        rTestPosTop;
		TPWrite "Side 1 A";
		MoveJ pSafeS1, vmax, fine, tWeldGun\WObj:=wobjSide1A200;
		!Code Goes Here
		MoveJ pSafeS181, vmax, fine, tWeldGun\WObj:=wobjSide1A200;
		SingArea\Wrist;
		MoveJ [[1183.18,1457.45,363.98],[0.0635628,0.517234,-0.779105,0.348461],[0,1,-3,1],[9E+09,9E+09,9E+09,9E+09,9E+09,9E+09]], vmax, z10, tWeldGun\WObj:=wobjSide1A200;
		MoveL [[1181.95,1536.61,-4.61],[0.0635699,0.51724,-0.779104,0.348453],[0,1,-2,1],[9E+09,9E+09,9E+09,9E+09,9E+09,9E+09]], v1000, z10, tWeldGun\WObj:=wobjSide1A200;
		ArcLStart [[1183.34,1532.14,-10.38],[0.0432656,0.526366,-0.780926,0.333501],[0,1,-2,1],[9E+09,9E+09,9E+09,9E+09,9E+09,9E+09]], v10, seam13, weld13\Weave:=weave1, fine, tWeldGun\WObj:=wobjSide1A200;
		ArcLEnd [[1206.22,1532.24,-10.36],[0.0432175,0.526382,-0.780937,0.333453],[0,1,-2,1],[9E+09,9E+09,9E+09,9E+09,9E+09,9E+09]], v10, seam13, weld13\Weave:=weave1, fine, tWeldGun\WObj:=wobjSide1A200;
		MoveL [[1204.62,1537.22,-4.87],[0.0635798,0.517232,-0.779109,0.348451],[0,1,-2,1],[9E+09,9E+09,9E+09,9E+09,9E+09,9E+09]], vmax, z10, tWeldGun\WObj:=wobjSide1A200;
		MoveL [[863.66,1538.85,77.89],[0.0635666,0.517243,-0.779097,0.348464],[0,1,-2,1],[9E+09,9E+09,9E+09,9E+09,9E+09,9E+09]], vmax, z10, tWeldGun\WObj:=wobjSide1A200;
		MoveJ [[861.58,1461.21,260.09],[0.14949,-0.376148,-0.839997,-0.361347],[0,1,-1,1],[9E+09,9E+09,9E+09,9E+09,9E+09,9E+09]], vmax, z10, tWeldGun\WObj:=wobjSide1A200;
		MoveL [[863.22,1468.67,-10.11],[0.149522,-0.376221,-0.839963,-0.361336],[0,1,-1,1],[9E+09,9E+09,9E+09,9E+09,9E+09,9E+09]], v1000, z10, tWeldGun\WObj:=wobjSide1A200;
		ArcLStart [[866.37,1476.97,-12.05],[0.0874714,-0.401117,-0.850564,-0.328626],[0,1,-1,1],[9E+09,9E+09,9E+09,9E+09,9E+09,9E+09]], v10, seam13, weld13\Weave:=weave1, fine, tWeldGun\WObj:=wobjSide1A200;
		ArcLEnd [[894.17,1477.17,-12.05],[0.0874956,-0.401178,-0.850524,-0.328648],[0,1,-1,1],[9E+09,9E+09,9E+09,9E+09,9E+09,9E+09]], v10, seam13, weld13\Weave:=weave1, fine, tWeldGun\WObj:=wobjSide1A200;
		MoveL [[886.08,1463.03,-7.28],[0.149478,-0.376156,-0.840008,-0.361317],[0,1,-1,1],[9E+09,9E+09,9E+09,9E+09,9E+09,9E+09]], vmax, z10, tWeldGun\WObj:=wobjSide1A200;
		MoveJ [[863.35,1506.96,224.59],[0.0635605,0.517248,-0.779091,0.348471],[0,1,-2,1],[9E+09,9E+09,9E+09,9E+09,9E+09,9E+09]], vmax, z10, tWeldGun\WObj:=wobjSide1A200;
		MoveL [[863.49,1538.37,-7.85],[0.0635592,0.51724,-0.779122,0.348415],[0,1,-2,1],[9E+09,9E+09,9E+09,9E+09,9E+09,9E+09]], vmax, z10, tWeldGun\WObj:=wobjSide1A200;
		ArcLStart [[859.58,1532.06,-11.51],[0.0485275,0.53765,-0.768469,0.343561],[0,1,-2,1],[9E+09,9E+09,9E+09,9E+09,9E+09,9E+09]], v10, seam13, weld13\Weave:=weave1, fine, tWeldGun\WObj:=wobjSide1A200;
		ArcLEnd [[891.59,1532.36,-10.59],[0.0487409,0.513057,-0.792225,0.326766],[0,1,-2,1],[9E+09,9E+09,9E+09,9E+09,9E+09,9E+09]], v10, seam13, weld13\Weave:=weave1, fine, tWeldGun\WObj:=wobjSide1A200;
		MoveL [[887.77,1539.90,182.89],[0.0635615,0.517251,-0.779088,0.348474],[0,1,-2,1],[9E+09,9E+09,9E+09,9E+09,9E+09,9E+09]], vmax, z10, tWeldGun\WObj:=wobjSide1A200;
		MoveJ [[1182.52,1470.34,61.27],[0.149538,-0.376243,-0.839941,-0.361358],[0,1,-1,1],[9E+09,9E+09,9E+09,9E+09,9E+09,9E+09]], vmax, z10, tWeldGun\WObj:=wobjSide1A200;
		MoveL [[1181.55,1464.42,-9.30],[0.148332,-0.500326,-0.790399,-0.320847],[0,1,-1,1],[9E+09,9E+09,9E+09,9E+09,9E+09,9E+09]], v1000, z10, tWeldGun\WObj:=wobjSide1A200;
		ArcLStart [[1177.33,1473.60,-12.87],[0.148345,-0.500351,-0.790382,-0.320842],[0,1,-1,1],[9E+09,9E+09,9E+09,9E+09,9E+09,9E+09]], v10, seam13, weld13\Weave:=weave1, fine, tWeldGun\WObj:=wobjSide1A200;
		ArcLEnd [[1207.54,1473.57,-12.86],[0.148337,-0.500345,-0.790386,-0.320845],[0,1,-1,1],[9E+09,9E+09,9E+09,9E+09,9E+09,9E+09]], v10, seam13, weld13\Weave:=weave1, fine, tWeldGun\WObj:=wobjSide1A200;
		MoveL [[1206.87,1462.04,-3.48],[0.148351,-0.500349,-0.790363,-0.320889],[0,1,-1,1],[9E+09,9E+09,9E+09,9E+09,9E+09,9E+09]], vmax, z10, tWeldGun\WObj:=wobjSide1A200;
		MoveL [[1203.94,921.98,77.52],[0.149416,-0.376356,-0.839957,-0.361252],[0,1,-1,1],[9E+09,9E+09,9E+09,9E+09,9E+09,9E+09]], vmax, z10, tWeldGun\WObj:=wobjSide1A200;
		MoveL [[1209.28,920.32,-0.95],[0.0811338,-0.402507,-0.844244,-0.344469],[0,1,-1,1],[9E+09,9E+09,9E+09,9E+09,9E+09,9E+09]], v1000, z10, tWeldGun\WObj:=wobjSide1A200;
		ArcLStart [[1208.91,928.66,-10.99],[0.081096,-0.402552,-0.84423,-0.344458],[0,1,-1,1],[9E+09,9E+09,9E+09,9E+09,9E+09,9E+09]], v10, seam13, weld13\Weave:=weave1, fine, tWeldGun\WObj:=wobjSide1A200;
		ArcLEnd [[1180.12,929.43,-11.01],[0.0811029,-0.402583,-0.844212,-0.344465],[0,1,0,1],[9E+09,9E+09,9E+09,9E+09,9E+09,9E+09]], v10, seam13, weld13\Weave:=weave1, fine, tWeldGun\WObj:=wobjSide1A200;
		MoveL [[1182.60,918.33,-2.85],[0.0811745,-0.402551,-0.844212,-0.344485],[0,1,0,1],[9E+09,9E+09,9E+09,9E+09,9E+09,9E+09]], vmax, z10, tWeldGun\WObj:=wobjSide1A200;
		MoveL [[883.71,921.14,-1.64],[0.149424,-0.37639,-0.839933,-0.361269],[0,1,0,1],[9E+09,9E+09,9E+09,9E+09,9E+09,9E+09]], vmax, z10, tWeldGun\WObj:=wobjSide1A200;
		MoveL [[891.05,920.87,-4.97],[0.15161,-0.376469,-0.855824,-0.320705],[0,1,-1,1],[9E+09,9E+09,9E+09,9E+09,9E+09,9E+09]], v1000, z10, tWeldGun\WObj:=wobjSide1A200;
		ArcLStart [[890.95,930.44,-12.87],[0.151512,-0.376481,-0.855837,-0.320703],[0,1,-1,1],[9E+09,9E+09,9E+09,9E+09,9E+09,9E+09]], v10, seam13, weld13\Weave:=weave1, fine, tWeldGun\WObj:=wobjSide1A200;
		ArcLEnd [[864.65,932.03,-12.68],[0.151535,-0.376589,-0.85577,-0.320744],[0,1,-1,1],[9E+09,9E+09,9E+09,9E+09,9E+09,9E+09]], v10, seam13, weld13\Weave:=weave1, fine, tWeldGun\WObj:=wobjSide1A200;
		MoveL [[866.54,921.07,-4.87],[0.151523,-0.376433,-0.855874,-0.320656],[0,1,-1,1],[9E+09,9E+09,9E+09,9E+09,9E+09,9E+09]], v100, z10, tWeldGun\WObj:=wobjSide1A200;
		MoveL [[861.26,919.79,117.88],[0.149443,-0.376442,-0.8399,-0.361285],[0,1,-1,1],[9E+09,9E+09,9E+09,9E+09,9E+09,9E+09]], vmax, z0, tWeldGun\WObj:=wobjSide1A200;
		MoveJ [[868.17,991.07,127.71],[0.0426372,-0.330552,0.858067,-0.39069],[0,1,-2,1],[9E+09,9E+09,9E+09,9E+09,9E+09,9E+09]], vmax, z0, tWeldGun\WObj:=wobjSide1A200;
		MoveL [[863.71,988.79,-2.92],[0.042941,-0.330682,0.857982,-0.390734],[0,0,-2,1],[9E+09,9E+09,9E+09,9E+09,9E+09,9E+09]], v1000, z10, tWeldGun\WObj:=wobjSide1A200;
		ArcLStart [[861.89,984.77,-9.70],[0.0429638,-0.330722,0.857953,-0.39076],[0,0,-2,1],[9E+09,9E+09,9E+09,9E+09,9E+09,9E+09]], v10, seam13, weld13\Weave:=weave1, fine, tWeldGun\WObj:=wobjSide1A200;
		ArcLEnd [[898.10,985.21,-7.50],[0.0432219,-0.327548,0.859798,-0.389348],[0,0,-2,1],[9E+09,9E+09,9E+09,9E+09,9E+09,9E+09]], v10, seam13, weld13\Weave:=weave1, fine, tWeldGun\WObj:=wobjSide1A200;
		MoveL [[889.59,992.71,-6.61],[0.0430178,-0.330607,0.858002,-0.390745],[0,0,-2,1],[9E+09,9E+09,9E+09,9E+09,9E+09,9E+09]], vmax, z10, tWeldGun\WObj:=wobjSide1A200;
		MoveL [[889.59,992.73,75.52],[0.0430306,-0.330621,0.857997,-0.390743],[0,1,-2,1],[9E+09,9E+09,9E+09,9E+09,9E+09,9E+09]], vmax, z10, tWeldGun\WObj:=wobjSide1A200;
		MoveL [[1177.66,992.72,75.52],[0.0430182,-0.33062,0.857997,-0.390745],[0,0,-2,1],[9E+09,9E+09,9E+09,9E+09,9E+09,9E+09]], vmax, z10, tWeldGun\WObj:=wobjSide1A200;
		MoveL [[1185.35,990.20,-3.61],[0.0429073,-0.330578,0.858028,-0.390724],[0,0,-2,1],[9E+09,9E+09,9E+09,9E+09,9E+09,9E+09]], v1000, z10, tWeldGun\WObj:=wobjSide1A200;
		ArcLStart [[1176.08,984.61,-10.65],[0.0451953,-0.325527,0.859941,-0.390503],[0,0,-2,1],[9E+09,9E+09,9E+09,9E+09,9E+09,9E+09]], v10, seam13, weld13\Weave:=weave1, fine, tWeldGun\WObj:=wobjSide1A200;
		ArcLEnd [[1210.47,984.70,-10.67],[0.0451959,-0.325517,0.859949,-0.390493],[0,0,-2,1],[9E+09,9E+09,9E+09,9E+09,9E+09,9E+09]], v10, seam13, weld13\Weave:=weave1, fine, tWeldGun\WObj:=wobjSide1A200;
		MoveL [[1208.39,990.70,-6.82],[0.0442447,-0.330375,0.858404,-0.389919],[0,0,-2,1],[9E+09,9E+09,9E+09,9E+09,9E+09,9E+09]], v1000, z10, tWeldGun\WObj:=wobjSide1A200;
		MoveL [[1207.95,989.04,392.36],[0.0429563,-0.330627,0.857995,-0.39075],[0,1,-2,1],[9E+09,9E+09,9E+09,9E+09,9E+09,9E+09]], vmax, z10, tWeldGun\WObj:=wobjSide1A200;
		MoveJ [[194.09,1536.38,108.42],[0.0907205,-0.623393,0.712906,0.308084],[0,-1,0,1],[9E+09,9E+09,9E+09,9E+09,9E+09,9E+09]], vmax, z10, tWeldGun\WObj:=wobjSide1A200;
		MoveL [[194.09,1534.55,21.51],[0.0907097,-0.623392,0.712903,0.308096],[0,-1,0,1],[9E+09,9E+09,9E+09,9E+09,9E+09,9E+09]], vmax, z10, tWeldGun\WObj:=wobjSide1A200;
		ArcLStart [[190.35,1535.97,0.59],[0.0903662,-0.623335,0.713039,0.307999],[0,-1,0,1],[9E+09,9E+09,9E+09,9E+09,9E+09,9E+09]], v20, seam13, weld13\Weave:=weave1, fine, tWeldGun\WObj:=wobjSide1A200;
		ArcLEnd [[159.94,1535.93,0.55],[0.090343,-0.623341,0.713041,0.307988],[0,-1,0,1],[9E+09,9E+09,9E+09,9E+09,9E+09,9E+09]], v20, seam13, weld13\Weave:=weave1, fine, tWeldGun\WObj:=wobjSide1A200;
		MoveL [[158.09,1532.35,8.43],[0.0907075,-0.623402,0.712898,0.30809],[0,-1,0,1],[9E+09,9E+09,9E+09,9E+09,9E+09,9E+09]], vmax, z10, tWeldGun\WObj:=wobjSide1A200;
		MoveL [[-128.01,1535.58,7.69],[0.090663,-0.623378,0.712945,0.308043],[1,0,0,1],[9E+09,9E+09,9E+09,9E+09,9E+09,9E+09]], vmax, z10, tWeldGun\WObj:=wobjSide1A200;
		ArcLStart [[-127.83,1537.58,1.69],[0.0906477,-0.623383,0.712936,0.308058],[1,0,0,1],[9E+09,9E+09,9E+09,9E+09,9E+09,9E+09]], v20, seam13, weld13\Weave:=weave1, fine, tWeldGun\WObj:=wobjSide1A200;
		ArcLEnd [[-163.90,1538.90,1.91],[0.0906267,-0.6234,0.712927,0.308051],[1,0,0,1],[9E+09,9E+09,9E+09,9E+09,9E+09,9E+09]], v20, seam13, weld13\Weave:=weave1, fine, tWeldGun\WObj:=wobjSide1A200;
		SingArea\Wrist;
		MoveL [[-158.90,1535.32,931.69],[0.0906389,-0.623348,0.712932,0.308139],[1,-2,1,0],[9E+09,9E+09,9E+09,9E+09,9E+09,9E+09]], vmax, z0, tWeldGun\WObj:=wobjSide1A200;
		MoveJ [[-173.66,614.72,251.09],[0.128906,0.0495871,0.95885,-0.248055],[1,-1,1,0],[9E+09,9E+09,9E+09,9E+09,9E+09,9E+09]], vmax, z0, tWeldGun\WObj:=wobjSide1A200;
		MoveL [[-145.55,555.68,15.34],[0.152232,0.0392509,0.96562,-0.207034],[1,-1,1,0],[9E+09,9E+09,9E+09,9E+09,9E+09,9E+09]], vmax, z0, tWeldGun\WObj:=wobjSide1A200;
		ArcLStart [[-145.25,553.61,5.23],[0.150684,0.0446148,0.957996,-0.239891],[1,-1,1,0],[9E+09,9E+09,9E+09,9E+09,9E+09,9E+09]], v20, seam13, weld13\Weave:=weave1, fine, tWeldGun\WObj:=wobjSide1A200;
		ArcLEnd [[-113.04,553.61,5.21],[0.150682,0.0446047,0.957994,-0.239902],[1,-1,1,0],[9E+09,9E+09,9E+09,9E+09,9E+09,9E+09]], v20, seam13, weld13\Weave:=weave1, fine, tWeldGun\WObj:=wobjSide1A200;
		MoveL [[-113.65,555.41,12.33],[0.152159,0.0393397,0.96563,-0.207027],[1,-1,1,0],[9E+09,9E+09,9E+09,9E+09,9E+09,9E+09]], vmax, z0, tWeldGun\WObj:=wobjSide1A200;
		MoveL [[173.88,557.63,12.23],[0.150918,0.0436625,0.959445,-0.234057],[1,-1,1,0],[9E+09,9E+09,9E+09,9E+09,9E+09,9E+09]], vmax, z0, tWeldGun\WObj:=wobjSide1A200;
		ArcLStart [[173.75,552.63,2.66],[0.150938,0.0436659,0.959441,-0.234061],[1,-1,1,0],[9E+09,9E+09,9E+09,9E+09,9E+09,9E+09]], v20, seam13, weld13\Weave:=weave1, fine, tWeldGun\WObj:=wobjSide1A200;
		ArcLEnd [[207.36,552.81,2.26],[0.150944,0.0436531,0.959435,-0.234083],[1,-1,1,0],[9E+09,9E+09,9E+09,9E+09,9E+09,9E+09]], v20, seam13, weld13\Weave:=weave1, fine, tWeldGun\WObj:=wobjSide1A200;
		MoveL [[207.49,559.40,13.87],[0.152119,0.0394488,0.965633,-0.20702],[1,-1,1,0],[9E+09,9E+09,9E+09,9E+09,9E+09,9E+09]], vmax, z0, tWeldGun\WObj:=wobjSide1A200;
		MoveL [[862.60,554.49,14.86],[0.152154,0.0392658,0.965627,-0.207055],[0,-2,1,0],[9E+09,9E+09,9E+09,9E+09,9E+09,9E+09]], vmax, z0, tWeldGun\WObj:=wobjSide1A200;
		ArcLStart [[864.91,549.07,1.34],[0.133495,0.0503347,0.954435,-0.262108],[0,-1,1,0],[9E+09,9E+09,9E+09,9E+09,9E+09,9E+09]], v20, seam13, weld13\Weave:=weave1, fine, tWeldGun\WObj:=wobjSide1A200;
		ArcLEnd [[899.31,549.07,1.33],[0.133493,0.0503325,0.954436,-0.262103],[0,-2,1,0],[9E+09,9E+09,9E+09,9E+09,9E+09,9E+09]], v20, seam13, weld13\Weave:=weave1, fine, tWeldGun\WObj:=wobjSide1A200;
		MoveL [[899.33,555.62,9.82],[0.152106,0.0393027,0.965639,-0.207029],[0,-2,1,0],[9E+09,9E+09,9E+09,9E+09,9E+09,9E+09]], vmax, z0, tWeldGun\WObj:=wobjSide1A200;
		MoveL [[1178.47,554.50,11.88],[0.149638,0.047924,0.952344,-0.261443],[0,-2,1,0],[9E+09,9E+09,9E+09,9E+09,9E+09,9E+09]], vmax, z0, tWeldGun\WObj:=wobjSide1A200;
		ArcLStart [[1182.61,548.27,-0.41],[0.119114,0.0614783,0.947533,-0.290197],[0,-2,1,0],[9E+09,9E+09,9E+09,9E+09,9E+09,9E+09]], v20, seam13, weld13\Weave:=weave1, fine, tWeldGun\WObj:=wobjSide1A200;
		ArcLEnd [[1211.37,548.80,-1.22],[0.119109,0.0614608,0.947531,-0.290208],[0,-2,1,0],[9E+09,9E+09,9E+09,9E+09,9E+09,9E+09]], v20, seam13, weld13\Weave:=weave1, fine, tWeldGun\WObj:=wobjSide1A200;
		MoveL [[1185.29,583.76,320.77],[0.152081,0.0394165,0.965666,-0.206898],[0,-2,1,0],[9E+09,9E+09,9E+09,9E+09,9E+09,9E+09]], vmax, z0, tWeldGun\WObj:=wobjSide1A200;
		MoveJ [[759.22,820.77,477.02],[0.128857,0.0495447,0.958803,-0.24827],[0,-1,1,0],[9E+09,9E+09,9E+09,9E+09,9E+09,9E+09]], vmax, z0, tWeldGun\WObj:=wobjSide1A200;
		!legs start here
		MoveJ [[-401.88,982.38,420.80],[0.377905,-0.177501,-0.908663,-0.00353082],[1,0,1,0],[9E+09,9E+09,9E+09,9E+09,9E+09,9E+09]], vmax, z0, tWeldGun;
		MoveL [[-401.87,982.37,-5.96],[0.377901,-0.177501,-0.908665,-0.00352363],[1,0,1,0],[9E+09,9E+09,9E+09,9E+09,9E+09,9E+09]], v1000, z0, tWeldGun;
		ArcLStart [[-404.58,981.09,-7.78],[0.37795,-0.177396,-0.908665,-0.00362024],[1,0,1,0],[9E+09,9E+09,9E+09,9E+09,9E+09,9E+09]], v10, seam13, weld13\Weave:=weave1, fine, tWeldGun;
		ArcL [[-403.34,957.35,-6.28],[0.377997,-0.177583,-0.90861,-0.00339797],[1,0,1,0],[9E+09,9E+09,9E+09,9E+09,9E+09,9E+09]], v10, seam13, weld13\Weave:=weave1, z10, tWeldGun;
		ArcLEnd [[-425.46,950.14,-7.20],[0.197405,-0.679804,-0.668803,-0.227157],[1,0,2,0],[9E+09,9E+09,9E+09,9E+09,9E+09,9E+09]], v10, seam13, weld13\Weave:=weave1, fine, tWeldGun;
		MoveL [[-425.48,941.74,3.95],[0.197405,-0.679809,-0.668795,-0.227167],[1,0,2,0],[9E+09,9E+09,9E+09,9E+09,9E+09,9E+09]], vmax, z0, tWeldGun;
		MoveL [[-432.39,895.03,94.24],[0.274951,-0.581467,-0.743558,-0.182811],[1,0,2,0],[9E+09,9E+09,9E+09,9E+09,9E+09,9E+09]], vmax, z0, tWeldGun;
		MoveL [[-1101.20,895.02,94.24],[0.274939,-0.581469,-0.743563,-0.182805],[1,0,2,0],[9E+09,9E+09,9E+09,9E+09,9E+09,9E+09]], vmax, z0, tWeldGun;
		MoveL [[-1101.70,938.01,-1.40],[0.240452,-0.654006,-0.686015,-0.209388],[1,0,2,0],[9E+09,9E+09,9E+09,9E+09,9E+09,9E+09]], v1000, z0, tWeldGun;
		ArcLStart [[-1102.46,946.94,-5.88],[0.240345,-0.654194,-0.685887,-0.20934],[1,0,2,0],[9E+09,9E+09,9E+09,9E+09,9E+09,9E+09]], v10, seam13, weld13\Weave:=weave1, fine, tWeldGun;
		ArcL [[-1122.33,944.31,-5.63],[0.240415,-0.654059,-0.68597,-0.209414],[1,0,2,0],[9E+09,9E+09,9E+09,9E+09,9E+09,9E+09]], v10, seam13, weld13\Weave:=weave1, z10, tWeldGun;
		ArcLEnd [[-1131.87,975.46,-7.21],[0.0370294,0.922956,0.0834677,0.373919],[1,0,3,0],[9E+09,9E+09,9E+09,9E+09,9E+09,9E+09]], v10, seam13, weld13\Weave:=weave1, fine, tWeldGun;
		MoveL [[-1142.99,977.01,6.44],[0.0501214,0.923455,0.0523108,0.376805],[1,0,3,0],[9E+09,9E+09,9E+09,9E+09,9E+09,9E+09]], vmax, z0, tWeldGun;
		MoveJ [[-1224.84,979.29,303.50],[0.0444685,0.923113,0.0666376,0.376092],[1,0,-1,0],[9E+09,9E+09,9E+09,9E+09,9E+09,9E+09]], vmax, z20, tWeldGun;
		MoveL [[-1198.60,1154.71,4.46],[0.0444461,0.923123,0.0666424,0.37607],[1,0,-1,0],[9E+09,9E+09,9E+09,9E+09,9E+09,9E+09]], v1000, z0, tWeldGun;
		ArcLStart [[-1190.33,1151.56,-7.20],[0.0443887,0.92316,0.0665763,0.375997],[1,0,-1,0],[9E+09,9E+09,9E+09,9E+09,9E+09,9E+09]], v10, seam13, weld13\Weave:=weave1, fine, tWeldGun;
		ArcL [[-1193.47,1177.01,-8.64],[0.0444674,0.923156,0.0665468,0.376002],[1,0,-1,0],[9E+09,9E+09,9E+09,9E+09,9E+09,9E+09]], v10, seam13, weld13\Weave:=weave1, z10, tWeldGun;
		ArcLEnd [[-1167.22,1193.43,-4.61],[0.211529,0.696313,-0.654269,0.205758],[1,-1,0,0],[9E+09,9E+09,9E+09,9E+09,9E+09,9E+09]], v10, seam13, weld13\Weave:=weave1, fine, tWeldGun;
		MoveL [[-1165.81,1197.81,-4.44],[0.289046,0.665942,-0.622199,0.292988],[1,0,0,0],[9E+09,9E+09,9E+09,9E+09,9E+09,9E+09]], vmax, z0, tWeldGun;
		MoveL [[-1167.37,1197.80,267.48],[0.269054,0.631082,-0.684208,0.247398],[1,-1,0,0],[9E+09,9E+09,9E+09,9E+09,9E+09,9E+09]], vmax, z0, tWeldGun;
		MoveJ [[-491.85,1197.38,267.48],[0.269045,0.631086,-0.684208,0.247399],[1,-1,0,0],[9E+09,9E+09,9E+09,9E+09,9E+09,9E+09]], vmax, z0, tWeldGun;
		MoveL [[-493.75,1206.46,4.64],[0.230361,0.671978,-0.666396,0.226485],[1,-1,0,0],[9E+09,9E+09,9E+09,9E+09,9E+09,9E+09]], v1000, z0, tWeldGun;
		ArcLStart [[-496.53,1197.25,-8.21],[0.230282,0.672061,-0.666354,0.226445],[1,-1,0,0],[9E+09,9E+09,9E+09,9E+09,9E+09,9E+09]], v10, seam13, weld13\Weave:=weave1, fine, tWeldGun;
		ArcL [[-474.00,1197.10,-7.28],[0.230378,0.67197,-0.666403,0.226474],[1,-1,0,0],[9E+09,9E+09,9E+09,9E+09,9E+09,9E+09]], v10, seam13, weld13\Weave:=weave1, z10, tWeldGun;
		ArcLEnd [[-464.66,1164.90,-10.34],[0.384973,0.00807935,-0.922617,-0.0225858],[1,-1,1,0],[9E+09,9E+09,9E+09,9E+09,9E+09,9E+09]], v10, seam13, weld13\Weave:=weave1, fine, tWeldGun;
		MoveL [[-460.21,1166.10,-6.29],[0.384934,0.00803439,-0.922633,-0.0226006],[1,-1,1,0],[9E+09,9E+09,9E+09,9E+09,9E+09,9E+09]], vmax, z5, tWeldGun;
		MoveL [[-460.61,1166.13,158.38],[0.384913,0.00804793,-0.922641,-0.0226089],[1,-1,1,0],[9E+09,9E+09,9E+09,9E+09,9E+09,9E+09]], vmax, z5, tWeldGun;
		MoveJ [[-411.67,714.00,66.77],[0.262804,0.646065,-0.670013,0.254199],[1,-1,0,0],[9E+09,9E+09,9E+09,9E+09,9E+09,9E+09]], vmax, z5, tWeldGun;
		MoveL [[-412.17,719.36,-3.08],[0.242994,0.661127,-0.665052,0.248138],[1,-1,0,0],[9E+09,9E+09,9E+09,9E+09,9E+09,9E+09]], vmax, z5, tWeldGun;
		ArcLStart [[-411.16,714.15,-3.03],[0.22013,0.668771,-0.676855,0.214842],[1,-1,0,0],[9E+09,9E+09,9E+09,9E+09,9E+09,9E+09]], v5, seam13, weld13\Weave:=weave1, fine, tWeldGun;
		ArcLEnd [[-430.39,714.15,-6.45],[0.220118,0.668773,-0.67685,0.214862],[1,-1,0,0],[9E+09,9E+09,9E+09,9E+09,9E+09,9E+09]], v5, seam13, weld13\Weave:=weave1, fine, tWeldGun;
		MoveL [[-433.52,712.50,86.63],[0.256209,0.656106,-0.660016,0.261269],[1,-1,0,0],[9E+09,9E+09,9E+09,9E+09,9E+09,9E+09]], vmax, z5, tWeldGun;
		MoveL [[-1103.37,713.70,123.92],[0.256219,0.656103,-0.660014,0.261271],[1,-1,0,0],[9E+09,9E+09,9E+09,9E+09,9E+09,9E+09]], vmax, z5, tWeldGun;
		MoveL [[-1103.35,717.29,-4.25],[0.256222,0.656097,-0.66001,0.261295],[1,-1,0,0],[9E+09,9E+09,9E+09,9E+09,9E+09,9E+09]], vmax, z5, tWeldGun;
		ArcLStart [[-1103.12,713.69,-5.87],[0.256215,0.656125,-0.659976,0.261315],[1,-1,0,0],[9E+09,9E+09,9E+09,9E+09,9E+09,9E+09]], v5, seam13, weld13\Weave:=weave1, fine, tWeldGun;
		ArcLEnd [[-1131.44,712.83,-4.90],[0.256552,0.655237,-0.660527,0.261822],[1,-1,0,0],[9E+09,9E+09,9E+09,9E+09,9E+09,9E+09]], v5, seam13, weld13\Weave:=weave1, fine, tWeldGun;
		MoveL [[-1209.09,671.31,55.31],[0.0790996,-0.947264,0.00476783,-0.310504],[1,-1,-1,0],[9E+09,9E+09,9E+09,9E+09,9E+09,9E+09]], vmax, z5, tWeldGun;
		MoveJ [[-1174.22,1417.20,153.64],[0.288404,-0.63354,-0.657568,-0.288193],[1,-1,-2,0],[9E+09,9E+09,9E+09,9E+09,9E+09,9E+09]], vmax, z5, tWeldGun;
		MoveL [[-1161.88,1424.25,9.40],[0.288254,-0.633648,-0.657559,-0.288125],[1,-1,-2,0],[9E+09,9E+09,9E+09,9E+09,9E+09,9E+09]], vmax, z5, tWeldGun;
		ArcLStart [[-1160.66,1428.75,-9.26],[0.26399,-0.634491,-0.667287,-0.287158],[1,-1,-2,0],[9E+09,9E+09,9E+09,9E+09,9E+09,9E+09]], v5, seam13, weld13\Weave:=weave1, fine, tWeldGun;
		ArcLEnd [[-1185.26,1428.75,-8.26],[0.263991,-0.634496,-0.667282,-0.287157],[1,-1,-2,0],[9E+09,9E+09,9E+09,9E+09,9E+09,9E+09]], v5, seam13, weld13\Weave:=weave1, fine, tWeldGun;
		MoveL [[-1308.95,1421.25,86.72],[0.288384,-0.633585,-0.657536,-0.288188],[1,-1,-2,0],[9E+09,9E+09,9E+09,9E+09,9E+09,9E+09]], vmax, z5, tWeldGun;
		MoveL [[-494.06,1426.01,134.66],[0.280642,-0.634844,-0.656104,-0.296212],[1,-1,-2,0],[9E+09,9E+09,9E+09,9E+09,9E+09,9E+09]], vmax, z5, tWeldGun;
		MoveL [[-492.29,1429.04,-11.80],[0.251506,-0.647279,-0.667794,-0.268007],[1,-1,-2,0],[9E+09,9E+09,9E+09,9E+09,9E+09,9E+09]], vmax, z5, tWeldGun;
		ArcLStart [[-491.87,1429.46,-11.99],[0.251491,-0.647295,-0.667791,-0.267988],[1,-1,-2,0],[9E+09,9E+09,9E+09,9E+09,9E+09,9E+09]], v5, seam13, weld13\Weave:=weave1, fine, tWeldGun;
		ArcLEnd [[-476.29,1430.44,-11.13],[0.251464,-0.647334,-0.667765,-0.267984],[1,-1,-2,0],[9E+09,9E+09,9E+09,9E+09,9E+09,9E+09]], v5, seam13, weld13\Weave:=weave1, fine, tWeldGun;
		MoveL [[-335.43,1418.41,452.48],[0.280609,-0.634847,-0.656145,-0.296146],[1,-1,-2,0],[9E+09,9E+09,9E+09,9E+09,9E+09,9E+09]], vmax, z5, tWeldGun;
		MoveJ pSafeS1, vmax, fine, tWeldGun;

	ENDPROC

    PROC rRUNSide1A300()
        VAR num i;
            !300 Gallon Space Saver
           	rTestPosTop;
		TPWrite "Side 1 A";
        MoveJ pSafeS1, vmax, fine, tWeldGun;


            FOR i FROM 1 TO WeldiiiCount DO

                ! Optional safety check
                IF wp300{i}.start.trans.x <> 0 THEN
                    RunWeld(i);
                ENDIF

            ENDFOR
		MoveJ pSafeS1, vmax, fine, tWeldGun;
	ENDPROC

	PROC ss_200()
           	rTestPosTop;
		TPWrite "Side 1 A";
		MoveJ pSafeS1, vmax, fine, tWeldGun;
		!Code Goes Here
		MoveJ pSafeS181, vmax, fine, tWeldGun;
		SingArea\Wrist;
		MoveJ [[1181.97,1536.60,299.24],[0.0635588,0.517232,-0.779106,0.348462],[0,1,-3,1],[9E+09,9E+09,9E+09,9E+09,9E+09,9E+09]], vmax, z10, tWeldGun;
		MoveL [[1181.96,1536.60,-12.62],[0.0635661,0.517237,-0.779104,0.348458],[0,1,-2,1],[9E+09,9E+09,9E+09,9E+09,9E+09,9E+09]], v1000, z10, tWeldGun;
		ArcLStart [[1181.53,1529.02,-11.65],[0.0635714,0.517237,-0.779104,0.348457],[0,1,-2,1],[9E+09,9E+09,9E+09,9E+09,9E+09,9E+09]], v10, seam13, weld13\Weave:=weave1, fine, tWeldGun;
		ArcLEnd [[1204.96,1529.87,-10.62],[0.0635614,0.517237,-0.779103,0.348461],[0,1,-2,1],[9E+09,9E+09,9E+09,9E+09,9E+09,9E+09]], v10, seam13, weld13\Weave:=weave1, fine, tWeldGun;
		MoveL [[1204.64,1537.23,-12.62],[0.0635617,0.517239,-0.7791,0.348464],[0,1,-2,1],[9E+09,9E+09,9E+09,9E+09,9E+09,9E+09]], vmax, z10, tWeldGun;
		MoveL [[863.66,1538.85,77.89],[0.0635666,0.517243,-0.779097,0.348464],[0,1,-2,1],[9E+09,9E+09,9E+09,9E+09,9E+09,9E+09]], vmax, z10, tWeldGun;
		MoveJ [[861.58,1461.21,260.09],[0.14949,-0.376148,-0.839997,-0.361347],[0,1,-1,1],[9E+09,9E+09,9E+09,9E+09,9E+09,9E+09]], vmax, z10, tWeldGun;
		MoveL [[863.23,1471.68,-11.89],[0.149517,-0.37621,-0.839967,-0.361342],[0,1,-1,1],[9E+09,9E+09,9E+09,9E+09,9E+09,9E+09]], v1000, z10, tWeldGun;
		ArcLStart [[863.88,1474.96,-12.64],[0.149558,-0.376296,-0.839897,-0.361396],[0,1,-1,1],[9E+09,9E+09,9E+09,9E+09,9E+09,9E+09]], v10, seam13, weld13\Weave:=weave1, fine, tWeldGun;
		ArcLEnd [[887.67,1475.21,-13.25],[0.149548,-0.376266,-0.839942,-0.361327],[0,1,-1,1],[9E+09,9E+09,9E+09,9E+09,9E+09,9E+09]], v10, seam13, weld13\Weave:=weave1, fine, tWeldGun;
		MoveL [[886.08,1463.03,-7.28],[0.149478,-0.376156,-0.840008,-0.361317],[0,1,-1,1],[9E+09,9E+09,9E+09,9E+09,9E+09,9E+09]], vmax, z10, tWeldGun;
		MoveJ [[863.35,1506.96,224.59],[0.0635605,0.517248,-0.779091,0.348471],[0,1,-2,1],[9E+09,9E+09,9E+09,9E+09,9E+09,9E+09]], vmax, z10, tWeldGun;
		MoveL [[863.21,1535.55,-10.64],[0.0635626,0.51725,-0.779093,0.348463],[0,1,-2,1],[9E+09,9E+09,9E+09,9E+09,9E+09,9E+09]], vmax, z10, tWeldGun;
		ArcLStart [[862.98,1531.20,-11.14],[0.0635851,0.517245,-0.779094,0.348464],[0,1,-2,1],[9E+09,9E+09,9E+09,9E+09,9E+09,9E+09]], v10, seam13, weld13\Weave:=weave1, fine, tWeldGun;
		ArcLEnd [[887.38,1530.81,-10.94],[0.0635922,0.517251,-0.779089,0.348465],[0,1,-2,1],[9E+09,9E+09,9E+09,9E+09,9E+09,9E+09]], v10, seam13, weld13\Weave:=weave1, fine, tWeldGun;
		MoveL [[887.77,1539.90,182.89],[0.0635615,0.517251,-0.779088,0.348474],[0,1,-2,1],[9E+09,9E+09,9E+09,9E+09,9E+09,9E+09]], vmax, z10, tWeldGun;
		MoveJ [[1182.52,1470.34,61.27],[0.149538,-0.376243,-0.839941,-0.361358],[0,1,-1,1],[9E+09,9E+09,9E+09,9E+09,9E+09,9E+09]], vmax, z10, tWeldGun;
		MoveL [[1182.53,1470.34,-16.07],[0.149529,-0.376231,-0.83995,-0.361353],[0,1,-1,1],[9E+09,9E+09,9E+09,9E+09,9E+09,9E+09]], v1000, z10, tWeldGun;
		ArcLStart [[1181.99,1475.51,-15.52],[0.149552,-0.376279,-0.83992,-0.361363],[0,1,-1,1],[9E+09,9E+09,9E+09,9E+09,9E+09,9E+09]], v10, seam13, weld13\Weave:=weave1, fine, tWeldGun;
		ArcLEnd [[1204.38,1476.47,-15.60],[0.149569,-0.376356,-0.839878,-0.361375],[0,1,-1,1],[9E+09,9E+09,9E+09,9E+09,9E+09,9E+09]], v10, seam13, weld13\Weave:=weave1, fine, tWeldGun;
		MoveL [[1202.33,1469.98,-15.09],[0.149549,-0.376274,-0.839922,-0.361365],[0,1,-1,1],[9E+09,9E+09,9E+09,9E+09,9E+09,9E+09]], vmax, z10, tWeldGun;
		MoveL [[1203.94,921.98,77.52],[0.149416,-0.376356,-0.839957,-0.361252],[0,1,-1,1],[9E+09,9E+09,9E+09,9E+09,9E+09,9E+09]], vmax, z10, tWeldGun;
		MoveL [[1203.94,921.99,-12.97],[0.149422,-0.376348,-0.839957,-0.361259],[0,1,-1,1],[9E+09,9E+09,9E+09,9E+09,9E+09,9E+09]], v1000, z10, tWeldGun;
		ArcLStart [[1203.94,928.79,-14.21],[0.149423,-0.376362,-0.839952,-0.361256],[0,1,-1,1],[9E+09,9E+09,9E+09,9E+09,9E+09,9E+09]], v10, seam13, weld13\Weave:=weave1, fine, tWeldGun;
		ArcLEnd [[1178.19,928.79,-14.21],[0.149422,-0.376442,-0.839904,-0.361285],[0,1,-1,1],[9E+09,9E+09,9E+09,9E+09,9E+09,9E+09]], v10, seam13, weld13\Weave:=weave1, fine, tWeldGun;
		MoveL [[1177.78,921.50,-1.65],[0.149422,-0.376364,-0.839949,-0.36126],[0,1,-1,1],[9E+09,9E+09,9E+09,9E+09,9E+09,9E+09]], vmax, z10, tWeldGun;
		MoveL [[883.71,921.14,-1.64],[0.149424,-0.37639,-0.839933,-0.361269],[0,1,0,1],[9E+09,9E+09,9E+09,9E+09,9E+09,9E+09]], vmax, z10, tWeldGun;
		MoveL [[883.71,926.93,-12.24],[0.149423,-0.3764,-0.839927,-0.361273],[0,0,0,1],[9E+09,9E+09,9E+09,9E+09,9E+09,9E+09]], v1000, z10, tWeldGun;
		ArcLStart [[885.40,928.75,-13.38],[0.149454,-0.376503,-0.839867,-0.361295],[0,0,0,1],[9E+09,9E+09,9E+09,9E+09,9E+09,9E+09]], v10, seam13, weld13\Weave:=weave1, fine, tWeldGun;
		ArcLEnd [[866.41,928.73,-13.39],[0.149444,-0.376494,-0.839881,-0.361275],[0,0,0,1],[9E+09,9E+09,9E+09,9E+09,9E+09,9E+09]], v10, seam13, weld13\Weave:=weave1, fine, tWeldGun;
		MoveL [[863.70,926.54,-12.25],[0.149435,-0.37642,-0.839913,-0.361282],[0,0,0,1],[9E+09,9E+09,9E+09,9E+09,9E+09,9E+09]], v100, z10, tWeldGun;
		MoveL [[861.26,919.79,117.88],[0.149443,-0.376442,-0.8399,-0.361285],[0,1,-1,1],[9E+09,9E+09,9E+09,9E+09,9E+09,9E+09]], vmax, z0, tWeldGun;
		MoveJ [[868.17,991.07,127.71],[0.0426372,-0.330552,0.858067,-0.39069],[0,1,-2,1],[9E+09,9E+09,9E+09,9E+09,9E+09,9E+09]], vmax, z0, tWeldGun;
		MoveL [[868.52,991.54,-9.45],[0.0429862,-0.330642,0.857997,-0.390729],[0,0,-2,1],[9E+09,9E+09,9E+09,9E+09,9E+09,9E+09]], v1000, z10, tWeldGun;
		ArcLStart [[865.93,978.35,-10.52],[0.0429801,-0.330651,0.857991,-0.390736],[0,0,-2,1],[9E+09,9E+09,9E+09,9E+09,9E+09,9E+09]], v10, seam13, weld13\Weave:=weave1, fine, tWeldGun;
		ArcLEnd [[888.37,978.36,-11.00],[0.0429914,-0.330695,0.857973,-0.390738],[0,0,-2,1],[9E+09,9E+09,9E+09,9E+09,9E+09,9E+09]], v10, seam13, weld13\Weave:=weave1, fine, tWeldGun;
		MoveL [[889.59,992.71,-9.41],[0.0430222,-0.330607,0.858002,-0.390746],[0,0,-2,1],[9E+09,9E+09,9E+09,9E+09,9E+09,9E+09]], vmax, z10, tWeldGun;
		MoveL [[889.59,992.73,75.52],[0.0430306,-0.330621,0.857997,-0.390743],[0,1,-2,1],[9E+09,9E+09,9E+09,9E+09,9E+09,9E+09]], vmax, z10, tWeldGun;
		MoveL [[1177.66,992.72,75.52],[0.0430182,-0.33062,0.857997,-0.390745],[0,0,-2,1],[9E+09,9E+09,9E+09,9E+09,9E+09,9E+09]], vmax, z10, tWeldGun;
		MoveL [[1185.41,992.70,-11.53],[0.0429716,-0.330606,0.858007,-0.390739],[0,0,-2,1],[9E+09,9E+09,9E+09,9E+09,9E+09,9E+09]], v1000, z10, tWeldGun;
		ArcLStart [[1180.66,978.10,-13.63],[0.0429557,-0.330625,0.857997,-0.390747],[0,0,-2,1],[9E+09,9E+09,9E+09,9E+09,9E+09,9E+09]], v10, seam13, weld13\Weave:=weave1, fine, tWeldGun;
		ArcLEnd [[1207.05,977.71,-13.62],[0.0429527,-0.330628,0.857994,-0.390751],[0,0,-2,1],[9E+09,9E+09,9E+09,9E+09,9E+09,9E+09]], v10, seam13, weld13\Weave:=weave1, fine, tWeldGun;
		MoveL [[1207.94,989.04,-11.16],[0.0429397,-0.330625,0.858002,-0.39074],[0,0,-2,1],[9E+09,9E+09,9E+09,9E+09,9E+09,9E+09]], v1000, z10, tWeldGun;
		MoveL [[1207.95,989.04,392.36],[0.0429563,-0.330627,0.857995,-0.39075],[0,1,-2,1],[9E+09,9E+09,9E+09,9E+09,9E+09,9E+09]], vmax, z10, tWeldGun;
		MoveJ [[194.09,1536.38,108.42],[0.0907205,-0.623393,0.712906,0.308084],[0,-1,0,1],[9E+09,9E+09,9E+09,9E+09,9E+09,9E+09]], vmax, z10, tWeldGun;
		MoveL [[194.09,1534.55,44.51],[0.0907126,-0.623398,0.712901,0.308089],[0,-1,0,1],[9E+09,9E+09,9E+09,9E+09,9E+09,9E+09]], vmax, z10, tWeldGun;
		ArcLStart [[191.25,1532.54,0.05],[0.0904838,-0.623408,0.712969,0.30798],[0,-1,0,1],[9E+09,9E+09,9E+09,9E+09,9E+09,9E+09]], v20, seam13, weld13\Weave:=weave1, fine, tWeldGun;
		ArcLEnd [[157.22,1532.54,0.51],[0.090482,-0.623409,0.712967,0.307981],[0,-1,0,1],[9E+09,9E+09,9E+09,9E+09,9E+09,9E+09]], v20, seam13, weld13\Weave:=weave1, fine, tWeldGun;
		MoveL [[158.09,1532.35,8.43],[0.0907075,-0.623402,0.712898,0.30809],[0,-1,0,1],[9E+09,9E+09,9E+09,9E+09,9E+09,9E+09]], vmax, z10, tWeldGun;
		MoveL [[-123.91,1535.35,12.43],[0.0907124,-0.623396,0.712903,0.308089],[1,0,0,1],[9E+09,9E+09,9E+09,9E+09,9E+09,9E+09]], vmax, z10, tWeldGun;
		ArcLStart [[-126.92,1534.33,1.43],[0.0907044,-0.623405,0.712895,0.308091],[1,0,0,1],[9E+09,9E+09,9E+09,9E+09,9E+09,9E+09]], v20, seam13, weld13\Weave:=weave1, fine, tWeldGun;
		ArcLEnd [[-160.92,1534.33,1.44],[0.090708,-0.623403,0.712896,0.308092],[1,0,0,1],[9E+09,9E+09,9E+09,9E+09,9E+09,9E+09]], v20, seam13, weld13\Weave:=weave1, fine, tWeldGun;
		MoveL [[-158.90,1535.32,931.69],[0.0906389,-0.623348,0.712932,0.308139],[1,-2,1,0],[9E+09,9E+09,9E+09,9E+09,9E+09,9E+09]], vmax, z0, tWeldGun;
		MoveJ [[-173.66,614.72,251.09],[0.128906,0.0495871,0.95885,-0.248055],[1,-1,1,0],[9E+09,9E+09,9E+09,9E+09,9E+09,9E+09]], vmax, z0, tWeldGun;
		MoveL [[-146.66,553.40,15.33],[0.15216,0.0393582,0.96563,-0.207021],[1,-1,1,0],[9E+09,9E+09,9E+09,9E+09,9E+09,9E+09]], vmax, z0, tWeldGun;
		ArcLStart [[-146.66,553.39,2.32],[0.152156,0.0393511,0.965628,-0.207036],[1,-1,1,0],[9E+09,9E+09,9E+09,9E+09,9E+09,9E+09]], v20, seam13, weld13\Weave:=weave1, fine, tWeldGun;
		ArcLEnd [[-114.67,554.39,1.31],[0.152148,0.0393507,0.965628,-0.207043],[1,-1,1,0],[9E+09,9E+09,9E+09,9E+09,9E+09,9E+09]], v20, seam13, weld13\Weave:=weave1, fine, tWeldGun;
		MoveL [[-113.65,555.41,12.33],[0.152159,0.0393397,0.96563,-0.207027],[1,-1,1,0],[9E+09,9E+09,9E+09,9E+09,9E+09,9E+09]], vmax, z0, tWeldGun;
		MoveL [[171.61,552.68,21.42],[0.152083,0.0394694,0.965633,-0.207041],[1,-1,1,0],[9E+09,9E+09,9E+09,9E+09,9E+09,9E+09]], vmax, z0, tWeldGun;
		ArcLStart [[171.63,552.69,-0.51],[0.152132,0.0394445,0.96562,-0.207073],[1,-1,1,0],[9E+09,9E+09,9E+09,9E+09,9E+09,9E+09]], v20, seam13, weld13\Weave:=weave1, fine, tWeldGun;
		ArcLEnd [[202.63,552.69,-0.52],[0.152129,0.0394303,0.965618,-0.207083],[1,-1,1,0],[9E+09,9E+09,9E+09,9E+09,9E+09,9E+09]], v20, seam13, weld13\Weave:=weave1, fine, tWeldGun;
		MoveL [[204.25,552.75,13.91],[0.152145,0.0394344,0.965619,-0.207068],[1,-1,1,0],[9E+09,9E+09,9E+09,9E+09,9E+09,9E+09]], vmax, z0, tWeldGun;
		MoveL [[860.18,549.11,14.83],[0.152112,0.039289,0.965636,-0.207043],[0,-2,1,0],[9E+09,9E+09,9E+09,9E+09,9E+09,9E+09]], vmax, z0, tWeldGun;
		ArcLStart [[860.21,550.17,-4.16],[0.152159,0.0392088,0.965632,-0.207039],[0,-2,1,0],[9E+09,9E+09,9E+09,9E+09,9E+09,9E+09]], v20, seam13, weld13\Weave:=weave1, fine, tWeldGun;
		ArcLEnd [[895.96,549.20,-3.18],[0.152141,0.039174,0.965634,-0.207051],[0,-2,1,0],[9E+09,9E+09,9E+09,9E+09,9E+09,9E+09]], v20, seam13, weld13\Weave:=weave1, fine, tWeldGun;
		MoveL [[895.37,549.34,9.83],[0.15211,0.0392827,0.965635,-0.207047],[0,-2,1,0],[9E+09,9E+09,9E+09,9E+09,9E+09,9E+09]], vmax, z0, tWeldGun;
		MoveL [[1175.32,546.94,11.83],[0.1496,0.0478929,0.95235,-0.261449],[0,-2,1,0],[9E+09,9E+09,9E+09,9E+09,9E+09,9E+09]], vmax, z0, tWeldGun;
		ArcLStart [[1177.31,546.94,-3.16],[0.149595,0.0478934,0.95235,-0.261454],[0,-2,1,0],[9E+09,9E+09,9E+09,9E+09,9E+09,9E+09]], v20, seam13, weld13\Weave:=weave1, fine, tWeldGun;
		ArcLEnd [[1209.31,546.95,-3.16],[0.149595,0.0478909,0.95235,-0.261454],[0,-2,1,0],[9E+09,9E+09,9E+09,9E+09,9E+09,9E+09]], v20, seam13, weld13\Weave:=weave1, fine, tWeldGun;
		MoveL [[1183.76,537.75,320.86],[0.152128,0.0394118,0.965637,-0.207003],[0,-2,1,0],[9E+09,9E+09,9E+09,9E+09,9E+09,9E+09]], vmax, z0, tWeldGun;
		MoveJ [[759.22,820.77,477.02],[0.128857,0.0495447,0.958803,-0.24827],[0,-1,1,0],[9E+09,9E+09,9E+09,9E+09,9E+09,9E+09]], vmax, z0, tWeldGun;
		MoveJ [[-401.88,982.38,420.80],[0.377905,-0.177501,-0.908663,-0.00353082],[1,0,1,0],[9E+09,9E+09,9E+09,9E+09,9E+09,9E+09]], vmax, z0, tWeldGun;
		MoveL [[-401.87,982.37,-5.96],[0.377901,-0.177501,-0.908665,-0.00352363],[1,0,1,0],[9E+09,9E+09,9E+09,9E+09,9E+09,9E+09]], v1000, z0, tWeldGun;
		ArcLStart [[-407.18,982.54,-5.95],[0.377941,-0.177364,-0.908675,-0.00361829],[1,0,1,0],[9E+09,9E+09,9E+09,9E+09,9E+09,9E+09]], v10, seam13, weld13\Weave:=weave1, fine, tWeldGun;
		ArcL [[-407.21,961.97,-7.34],[0.377917,-0.177516,-0.908656,-0.00352015],[1,0,1,0],[9E+09,9E+09,9E+09,9E+09,9E+09,9E+09]], v10, seam13, weld13\Weave:=weave1, z10, tWeldGun;
		ArcLEnd [[-429.48,955.83,-6.96],[0.274941,-0.581479,-0.743555,-0.1828],[1,0,2,0],[9E+09,9E+09,9E+09,9E+09,9E+09,9E+09]], v10, seam13, weld13\Weave:=weave1, fine, tWeldGun;
		MoveL [[-432.47,945.01,-6.78],[0.274937,-0.581449,-0.743579,-0.182803],[1,0,2,0],[9E+09,9E+09,9E+09,9E+09,9E+09,9E+09]], vmax, z0, tWeldGun;
		MoveL [[-432.39,895.03,94.24],[0.274951,-0.581467,-0.743558,-0.182811],[1,0,2,0],[9E+09,9E+09,9E+09,9E+09,9E+09,9E+09]], vmax, z0, tWeldGun;
		MoveL [[-1101.20,895.02,94.24],[0.274939,-0.581469,-0.743563,-0.182805],[1,0,2,0],[9E+09,9E+09,9E+09,9E+09,9E+09,9E+09]], vmax, z0, tWeldGun;
		MoveL [[-1101.21,942.37,-3.25],[0.274946,-0.581512,-0.743526,-0.182807],[1,0,2,0],[9E+09,9E+09,9E+09,9E+09,9E+09,9E+09]], v1000, z0, tWeldGun;
		ArcLStart [[-1099.81,952.01,-6.02],[0.23841,-0.593999,-0.734594,-0.225162],[1,0,2,0],[9E+09,9E+09,9E+09,9E+09,9E+09,9E+09]], v10, seam13, weld13\Weave:=weave1, fine, tWeldGun;
		ArcL [[-1121.08,951.80,-5.63],[0.238289,-0.634044,-0.696044,-0.238181],[1,0,2,0],[9E+09,9E+09,9E+09,9E+09,9E+09,9E+09]], v10, seam13, weld13\Weave:=weave1, z10, tWeldGun;
		ArcLEnd [[-1129.28,975.89,-6.00],[0.0369776,0.92297,0.0835389,0.373873],[1,0,3,0],[9E+09,9E+09,9E+09,9E+09,9E+09,9E+09]], v10, seam13, weld13\Weave:=weave1, fine, tWeldGun;
		MoveL [[-1142.99,977.01,6.44],[0.0501214,0.923455,0.0523108,0.376805],[1,0,3,0],[9E+09,9E+09,9E+09,9E+09,9E+09,9E+09]], vmax, z0, tWeldGun;
		MoveJ [[-1142.58,979.31,303.50],[0.0444513,0.923112,0.0666342,0.376096],[1,0,-1,0],[9E+09,9E+09,9E+09,9E+09,9E+09,9E+09]], vmax, z20, tWeldGun;
		MoveL [[-1192.76,1156.53,-4.42],[0.044443,0.923122,0.0666432,0.376072],[1,0,-1,0],[9E+09,9E+09,9E+09,9E+09,9E+09,9E+09]], v1000, z0, tWeldGun;
		ArcLStart [[-1192.23,1155.72,-3.63],[0.0444473,0.923132,0.0666323,0.376048],[1,0,-1,0],[9E+09,9E+09,9E+09,9E+09,9E+09,9E+09]], v10, seam13, weld13\Weave:=weave1, fine, tWeldGun;
		ArcL [[-1191.71,1175.69,-5.33],[0.0444379,0.923126,0.0666324,0.376065],[1,0,-1,0],[9E+09,9E+09,9E+09,9E+09,9E+09,9E+09]], v10, seam13, weld13\Weave:=weave1, z10, tWeldGun;
		ArcLEnd [[-1165.81,1187.00,-4.44],[0.28905,0.665936,-0.622204,0.292989],[1,0,0,0],[9E+09,9E+09,9E+09,9E+09,9E+09,9E+09]], v10, seam13, weld13\Weave:=weave1, fine, tWeldGun;
		MoveL [[-1165.81,1197.81,-4.44],[0.289046,0.665942,-0.622199,0.292988],[1,0,0,0],[9E+09,9E+09,9E+09,9E+09,9E+09,9E+09]], vmax, z0, tWeldGun;
		MoveL [[-1167.37,1197.80,267.48],[0.269054,0.631082,-0.684208,0.247398],[1,-1,0,0],[9E+09,9E+09,9E+09,9E+09,9E+09,9E+09]], vmax, z0, tWeldGun;
		MoveJ [[-491.85,1197.38,267.48],[0.269045,0.631086,-0.684208,0.247399],[1,-1,0,0],[9E+09,9E+09,9E+09,9E+09,9E+09,9E+09]], vmax, z0, tWeldGun;
		MoveL [[-495.49,1197.07,-6.30],[0.260132,0.661057,-0.654909,0.257739],[1,-1,0,0],[9E+09,9E+09,9E+09,9E+09,9E+09,9E+09]], v1000, z0, tWeldGun;
		ArcLStart [[-495.49,1192.07,-6.30],[0.260133,0.661061,-0.654906,0.257736],[1,-1,0,0],[9E+09,9E+09,9E+09,9E+09,9E+09,9E+09]], v10, seam13, weld13\Weave:=weave1, fine, tWeldGun;
		ArcL [[-474.53,1190.57,-6.48],[0.263861,0.655019,-0.660957,0.253897],[1,-1,0,0],[9E+09,9E+09,9E+09,9E+09,9E+09,9E+09]], v10, seam13, weld13\Weave:=weave1, z10, tWeldGun;
		ArcLEnd [[-467.21,1164.88,-8.10],[0.384925,0.00804232,-0.922637,-0.0225898],[1,-1,1,0],[9E+09,9E+09,9E+09,9E+09,9E+09,9E+09]], v10, seam13, weld13\Weave:=weave1, fine, tWeldGun;
		MoveL [[-460.21,1166.10,-6.29],[0.384934,0.00803439,-0.922633,-0.0226006],[1,-1,1,0],[9E+09,9E+09,9E+09,9E+09,9E+09,9E+09]], vmax, z5, tWeldGun;
		MoveL [[-460.61,1166.12,771.55],[0.384916,0.00803537,-0.92264,-0.0226078],[1,-1,1,0],[9E+09,9E+09,9E+09,9E+09,9E+09,9E+09]], vmax, z5, tWeldGun;
		MoveJ pSafeS1, vmax, fine, tWeldGun;
	ENDPROC

	PROC rRUNSIDE1A100()
		MoveJ [[895.91,925.45,959.23],[0.222593,0.0151737,0.948305,-0.225698],[0,-1,0,0],[9E+09,9E+09,9E+09,9E+09,9E+09,9E+09]], vmax, z50, tWeldGun\WObj:=wobjSide1A200;
		MoveJ [[1169.38,1081.61,325.39],[0.296115,-0.947077,-0.052822,0.112127],[0,-2,0,1],[9E+09,9E+09,9E+09,9E+09,9E+09,9E+09]], vmax, z50, tWeldGun;
		MoveL [[1189.01,1078.57,4.64],[0.333702,-0.921867,0.118424,-0.157418],[0,-2,-1,1],[9E+09,9E+09,9E+09,9E+09,9E+09,9E+09]], v1000, z50, tWeldGun;
		ArcLStart [[1185.61,1080.58,-9.86],[0.333643,-0.921896,0.118528,-0.157299],[0,-2,-1,1],[9E+09,9E+09,9E+09,9E+09,9E+09,9E+09]], v10, seam13, weld13\Weave:=weave1, fine, tWeldGun;
		ArcLEnd [[1153.22,1080.55,-9.89],[0.333626,-0.921901,0.118526,-0.157301],[0,-2,-1,1],[9E+09,9E+09,9E+09,9E+09,9E+09,9E+09]], v10, seam13, weld13\Weave:=weave1, fine, tWeldGun;
		MoveL [[1157.55,1079.96,5.67],[0.333709,-0.921874,0.118398,-0.157383],[0,-2,-1,1],[9E+09,9E+09,9E+09,9E+09,9E+09,9E+09]], vmax, z5, tWeldGun;
		MoveL [[864.56,1073.01,5.26],[0.379695,-0.916748,-0.042496,0.116617],[0,-2,-1,1],[9E+09,9E+09,9E+09,9E+09,9E+09,9E+09]], vmax, z5, tWeldGun;
		ArcLStart [[862.19,1074.19,-3.35],[0.379691,-0.916749,-0.0424859,0.116625],[0,-2,-1,1],[9E+09,9E+09,9E+09,9E+09,9E+09,9E+09]], v10, seam13, weld13\Weave:=weave1, fine, tWeldGun;
		ArcLEnd [[831.24,1074.23,-3.33],[0.379713,-0.916742,-0.0424399,0.116624],[0,-2,-1,1],[9E+09,9E+09,9E+09,9E+09,9E+09,9E+09]], v10, seam13, weld13\Weave:=weave1, fine, tWeldGun;
		MoveL [[834.56,1075.21,12.06],[0.379682,-0.916754,-0.0425092,0.116603],[0,-2,-1,1],[9E+09,9E+09,9E+09,9E+09,9E+09,9E+09]], vmax, z5, tWeldGun;
		MoveL [[172.30,1074.14,5.27],[0.379642,-0.916784,-0.0424626,0.11652],[0,-2,-1,1],[9E+09,9E+09,9E+09,9E+09,9E+09,9E+09]], vmax, z5, tWeldGun;
		ArcLStart [[172.45,1077.16,-3.73],[0.37965,-0.916783,-0.042437,0.116513],[0,-2,-1,1],[9E+09,9E+09,9E+09,9E+09,9E+09,9E+09]], v10, seam13, weld13\Weave:=weave1, fine, tWeldGun;
		ArcLEnd [[141.11,1075.63,-6.35],[0.394237,-0.896713,-0.191368,0.0621412],[0,-2,-1,1],[9E+09,9E+09,9E+09,9E+09,9E+09,9E+09]], v10, seam13, weld13\Weave:=weave1, fine, tWeldGun;
		MoveL [[141.10,1062.84,1.66],[0.394214,-0.896726,-0.191336,0.0621991],[0,-2,-1,1],[9E+09,9E+09,9E+09,9E+09,9E+09,9E+09]], vmax, z5, tWeldGun;
		MoveL [[-144.86,1070.65,3.80],[0.337591,-0.932768,-0.0489574,0.116536],[0,-2,-1,1],[9E+09,9E+09,9E+09,9E+09,9E+09,9E+09]], vmax, z5, tWeldGun;
		ArcLStart [[-144.83,1077.50,-2.20],[0.337605,-0.932765,-0.048953,0.116519],[0,-2,-1,1],[9E+09,9E+09,9E+09,9E+09,9E+09,9E+09]], v10, seam13, weld13\Weave:=weave1, fine, tWeldGun;
		ArcLEnd [[-176.80,1077.27,-2.42],[0.337568,-0.932779,-0.0489017,0.116534],[0,-2,-1,1],[9E+09,9E+09,9E+09,9E+09,9E+09,9E+09]], v10, seam13, weld13\Weave:=weave1, fine, tWeldGun;
		SingArea\Wrist;
		MoveL [[-200.44,1085.42,415.26],[0.379667,-0.916774,-0.042596,0.116465],[0,-2,-1,1],[9E+09,9E+09,9E+09,9E+09,9E+09,9E+09]], vmax, z5, tWeldGun;
		MoveJ [[-173.57,559.75,42.74],[0.145109,0.845875,-0.418866,0.296634],[1,0,-1,0],[9E+09,9E+09,9E+09,9E+09,9E+09,9E+09]], vmax, z5, tWeldGun;
		MoveL [[-170.35,568.46,-5.16],[0.145203,0.845842,-0.418973,0.29653],[1,0,-1,0],[9E+09,9E+09,9E+09,9E+09,9E+09,9E+09]], vmax, z5, tWeldGun;
		ArcLStart [[-170.35,561.67,-11.54],[0.145203,0.845851,-0.418953,0.296532],[1,0,-1,0],[9E+09,9E+09,9E+09,9E+09,9E+09,9E+09]], v10, seam13, weld13\Weave:=weave1, fine, tWeldGun;
		ArcLEnd [[-141.78,561.68,-11.54],[0.145216,0.845844,-0.418977,0.296513],[1,0,-1,0],[9E+09,9E+09,9E+09,9E+09,9E+09,9E+09]], v10, seam13, weld13\Weave:=weave1, fine, tWeldGun;
		MoveL [[-135.50,566.77,5.60],[0.145085,0.84588,-0.41892,0.296555],[1,0,-1,0],[9E+09,9E+09,9E+09,9E+09,9E+09,9E+09]], vmax, z5, tWeldGun;
		MoveL [[151.70,563.89,2.38],[0.145279,0.845821,-0.418979,0.296543],[0,0,-1,0],[9E+09,9E+09,9E+09,9E+09,9E+09,9E+09]], vmax, z5, tWeldGun;
		ArcLStart [[147.91,561.67,-12.61],[0.145298,0.845824,-0.41896,0.296552],[0,0,-1,0],[9E+09,9E+09,9E+09,9E+09,9E+09,9E+09]], v10, seam13, weld13\Weave:=weave1, fine, tWeldGun;
		ArcLEnd [[179.68,561.61,-12.60],[0.145306,0.845823,-0.418965,0.296545],[0,0,-1,0],[9E+09,9E+09,9E+09,9E+09,9E+09,9E+09]], v10, seam13, weld13\Weave:=weave1, fine, tWeldGun;
		MoveL [[179.70,567.65,-1.58],[0.145437,0.845826,-0.418906,0.296553],[0,0,-1,0],[9E+09,9E+09,9E+09,9E+09,9E+09,9E+09]], vmax, z5, tWeldGun;
		MoveL [[838.33,565.65,0.78],[0.145096,0.845788,-0.419047,0.296632],[0,0,-2,0],[9E+09,9E+09,9E+09,9E+09,9E+09,9E+09]], vmax, z5, tWeldGun;
		ArcLStart [[837.91,559.63,-15.44],[0.14512,0.845784,-0.419056,0.29662],[0,0,-2,0],[9E+09,9E+09,9E+09,9E+09,9E+09,9E+09]], v10, seam13, weld13\Weave:=weave1, fine, tWeldGun;
		ArcLEnd [[868.85,559.41,-15.48],[0.145145,0.845802,-0.419023,0.296601],[0,0,-2,0],[9E+09,9E+09,9E+09,9E+09,9E+09,9E+09]], v10, seam13, weld13\Weave:=weave1, fine, tWeldGun;
		MoveL [[869.08,565.56,-7.05],[0.145032,0.845778,-0.419043,0.296696],[0,0,-2,0],[9E+09,9E+09,9E+09,9E+09,9E+09,9E+09]], vmax, z5, tWeldGun;
		MoveL [[1154.26,567.31,-2.43],[0.145055,0.845814,-0.419044,0.296583],[0,0,-2,0],[9E+09,9E+09,9E+09,9E+09,9E+09,9E+09]], vmax, z5, tWeldGun;
		ArcLStart [[1154.25,559.10,-16.64],[0.145066,0.845816,-0.419041,0.296576],[0,0,-2,0],[9E+09,9E+09,9E+09,9E+09,9E+09,9E+09]], v10, seam13, weld13\Weave:=weave1, fine, tWeldGun;
		ArcLEnd [[1186.24,558.29,-16.04],[0.145087,0.845809,-0.419057,0.296562],[0,0,-2,0],[9E+09,9E+09,9E+09,9E+09,9E+09,9E+09]], v10, seam13, weld13\Weave:=weave1, fine, tWeldGun;
		MoveL [[1189.43,560.09,663.81],[0.145007,0.845796,-0.418995,0.296726],[0,0,-2,0],[9E+09,9E+09,9E+09,9E+09,9E+09,9E+09]], vmax, z5, tWeldGun;
		MoveJ [[-229.23,1115.81,554.88],[0.237488,0.691166,-0.628837,0.265431],[1,-1,-4,0],[9E+09,9E+09,9E+09,9E+09,9E+09,9E+09]], vmax, z5, tWeldGun;
		MoveL [[-412.06,717.19,27.71],[0.270403,0.66951,-0.638814,0.265624],[1,0,-4,0],[9E+09,9E+09,9E+09,9E+09,9E+09,9E+09]], vmax, z5, tWeldGun;
		MoveL [[-413.84,720.92,-0.46],[0.249904,0.677081,-0.652542,0.230865],[1,-1,-4,0],[9E+09,9E+09,9E+09,9E+09,9E+09,9E+09]], vmax, z5, tWeldGun;
		ArcLStart [[-413.85,715.51,-6.45],[0.249932,0.67707,-0.652544,0.230859],[1,-1,-4,0],[9E+09,9E+09,9E+09,9E+09,9E+09,9E+09]], v5, seam13, weld13\Weave:=weave1, fine, tWeldGun;
		ArcLEnd [[-433.02,715.70,-6.65],[0.249921,0.677092,-0.652516,0.230888],[1,-1,-4,0],[9E+09,9E+09,9E+09,9E+09,9E+09,9E+09]], v5, seam13, weld13\Weave:=weave1, fine, tWeldGun;
		MoveL [[-433.02,721.69,79.27],[0.249938,0.677071,-0.652532,0.230886],[1,-1,-4,0],[9E+09,9E+09,9E+09,9E+09,9E+09,9E+09]], vmax, z5, tWeldGun;
		MoveL [[-1100.50,721.09,94.11],[0.270393,0.669535,-0.638788,0.265635],[1,-1,-4,0],[9E+09,9E+09,9E+09,9E+09,9E+09,9E+09]], vmax, z5, tWeldGun;
		MoveL [[-1103.19,722.45,8.00],[0.239603,0.681202,-0.652992,0.228379],[1,-1,-4,0],[9E+09,9E+09,9E+09,9E+09,9E+09,9E+09]], vmax, z5, tWeldGun;
		ArcLStart [[-1103.19,713.56,-5.56],[0.239599,0.681202,-0.652993,0.228381],[1,-1,-4,0],[9E+09,9E+09,9E+09,9E+09,9E+09,9E+09]], v5, seam13, weld13\Weave:=weave1, fine, tWeldGun;
		ArcLEnd [[-1123.14,713.55,-4.77],[0.239595,0.681192,-0.652991,0.228416],[1,-1,-4,0],[9E+09,9E+09,9E+09,9E+09,9E+09,9E+09]], v5, seam13, weld13\Weave:=weave1, fine, tWeldGun;
		MoveL [[-1124.97,712.38,115.49],[0.270384,0.669531,-0.638781,0.26567],[1,-1,-4,0],[9E+09,9E+09,9E+09,9E+09,9E+09,9E+09]], vmax, z5, tWeldGun;
		MoveJ [[-1119.62,941.62,98.59],[0.263153,-0.665669,-0.65042,-0.254146],[1,0,-2,0],[9E+09,9E+09,9E+09,9E+09,9E+09,9E+09]], vmax, z5, tWeldGun;
		MoveL [[-1103.53,941.47,2.67],[0.263185,-0.665692,-0.650383,-0.254147],[1,0,-2,0],[9E+09,9E+09,9E+09,9E+09,9E+09,9E+09]], vmax, z5, tWeldGun;
		ArcLStart [[-1102.50,948.16,-6.90],[0.245378,-0.666002,-0.671984,-0.211351],[1,0,-2,0],[9E+09,9E+09,9E+09,9E+09,9E+09,9E+09]], v5, seam13, weld13\Weave:=weave1, fine, tWeldGun;
		ArcL [[-1124.20,945.08,-8.53],[0.241268,-0.666756,-0.672776,-0.211185],[1,0,-2,0],[9E+09,9E+09,9E+09,9E+09,9E+09,9E+09]], v5, seam13, weld13\Weave:=weave1, z10, tWeldGun;
		ArcLEnd [[-1132.51,978.64,-7.54],[0.0250689,0.926224,0.0082503,0.376049],[1,0,-1,0],[9E+09,9E+09,9E+09,9E+09,9E+09,9E+09]], v5, seam13, weld13\Weave:=weave1, fine, tWeldGun;
		MoveL [[-1148.62,985.17,63.09],[0.0198579,0.898733,0.00249179,0.438039],[1,-1,-1,0],[9E+09,9E+09,9E+09,9E+09,9E+09,9E+09]], vmax, z5, tWeldGun;
		MoveL [[-1199.14,1157.80,50.93],[0.0198608,0.898743,0.00250084,0.43802],[1,-1,-1,0],[9E+09,9E+09,9E+09,9E+09,9E+09,9E+09]], vmax, z5, tWeldGun;
		MoveL [[-1195.49,1156.64,0.22],[0.0202314,0.914596,0.00160063,0.403859],[1,0,-1,0],[9E+09,9E+09,9E+09,9E+09,9E+09,9E+09]], vmax, z5, tWeldGun;
		ArcLStart [[-1192.13,1157.24,-7.56],[0.0202377,0.91461,0.00159549,0.403829],[1,0,-1,0],[9E+09,9E+09,9E+09,9E+09,9E+09,9E+09]], v5, seam13, weld13\Weave:=weave1, fine, tWeldGun;
		ArcL [[-1195.11,1177.16,-6.96],[0.0243873,0.92589,-0.000794778,0.377005],[1,0,-1,0],[9E+09,9E+09,9E+09,9E+09,9E+09,9E+09]], v5, seam13, weld13\Weave:=weave1, z10, tWeldGun;
		ArcLEnd [[-1166.64,1194.35,-4.47],[0.234917,0.673253,-0.666667,0.217024],[1,-1,0,0],[9E+09,9E+09,9E+09,9E+09,9E+09,9E+09]], v5, seam13, weld13\Weave:=weave1, fine, tWeldGun;
		MoveL [[-1164.13,1200.44,93.33],[0.251271,0.657126,-0.66952,0.23831],[1,-1,0,0],[9E+09,9E+09,9E+09,9E+09,9E+09,9E+09]], vmax, z5, tWeldGun;
		MoveJ [[-1176.39,1428.24,109.35],[0.303454,-0.641239,-0.63752,-0.300495],[1,-1,2,0],[9E+09,9E+09,9E+09,9E+09,9E+09,9E+09]], vmax, z5, tWeldGun;
		MoveL [[-1186.42,1420.24,9.09],[0.262683,-0.660481,-0.654281,-0.258224],[1,0,2,0],[9E+09,9E+09,9E+09,9E+09,9E+09,9E+09]], vmax, z5, tWeldGun;
		ArcLStart [[-1183.89,1427.01,-5.32],[0.262685,-0.660493,-0.654268,-0.258224],[1,0,2,0],[9E+09,9E+09,9E+09,9E+09,9E+09,9E+09]], v30, seam13, weld13\Weave:=weave1, fine, tWeldGun;
		ArcLEnd [[-1164.71,1427.19,-6.55],[0.262711,-0.66047,-0.654286,-0.258211],[1,0,2,0],[9E+09,9E+09,9E+09,9E+09,9E+09,9E+09]], v5, seam13, weld13\Weave:=weave1, fine, tWeldGun;
		MoveL [[-1165.10,1427.68,74.68],[0.262682,-0.660472,-0.654289,-0.258226],[1,0,2,0],[9E+09,9E+09,9E+09,9E+09,9E+09,9E+09]], vmax, z5, tWeldGun;
		MoveL [[-495.20,1424.53,122.41],[0.28862,-0.64963,-0.643265,-0.284411],[1,-1,2,0],[9E+09,9E+09,9E+09,9E+09,9E+09,9E+09]], vmax, z5, tWeldGun;
		MoveL [[-492.11,1424.64,-4.56],[0.230632,-0.671635,-0.668577,-0.220728],[1,0,2,0],[9E+09,9E+09,9E+09,9E+09,9E+09,9E+09]], vmax, z5, tWeldGun;
		ArcLStart [[-494.82,1430.84,-11.36],[0.230629,-0.671668,-0.668546,-0.220726],[1,0,2,0],[9E+09,9E+09,9E+09,9E+09,9E+09,9E+09]], v5, seam13, weld13\Weave:=weave1, fine, tWeldGun;
		ArcLEnd [[-475.00,1430.64,-11.57],[0.230621,-0.671683,-0.668534,-0.220724],[1,0,2,0],[9E+09,9E+09,9E+09,9E+09,9E+09,9E+09]], v5, seam13, weld13\Weave:=weave1, fine, tWeldGun;
		MoveL [[-474.63,1411.30,125.45],[0.288602,-0.649679,-0.643225,-0.284408],[1,-1,2,0],[9E+09,9E+09,9E+09,9E+09,9E+09,9E+09]], vmax, z5, tWeldGun;
		MoveJ [[-479.04,1241.31,118.19],[0.268582,0.650118,-0.664304,0.252806],[1,-1,0,0],[9E+09,9E+09,9E+09,9E+09,9E+09,9E+09]], vmax, z5, tWeldGun;
		MoveL [[-495.83,1201.80,-1.90],[0.268594,0.650121,-0.6643,0.252797],[1,-1,0,0],[9E+09,9E+09,9E+09,9E+09,9E+09,9E+09]], vmax, z5, tWeldGun;
		ArcLStart [[-494.84,1196.21,-9.49],[0.268603,0.650127,-0.664292,0.252793],[1,-1,0,0],[9E+09,9E+09,9E+09,9E+09,9E+09,9E+09]], v5, seam13, weld13\Weave:=weave1, fine, tWeldGun;
		ArcL [[-476.48,1196.50,-9.26],[0.268632,0.650097,-0.664312,0.252787],[1,-1,0,0],[9E+09,9E+09,9E+09,9E+09,9E+09,9E+09]], v5, seam13, weld13\Weave:=weave1, z10, tWeldGun;
		ArcLEnd [[-465.51,1166.36,-12.09],[0.390509,0.0535053,-0.919043,-0.000194166],[1,-1,1,0],[9E+09,9E+09,9E+09,9E+09,9E+09,9E+09]], v5, seam13, weld13\Weave:=weave1, fine, tWeldGun;
		MoveL [[-435.96,1164.94,59.58],[0.390502,0.0535497,-0.919044,-0.000186584],[1,-1,1,0],[9E+09,9E+09,9E+09,9E+09,9E+09,9E+09]], vmax, z5, tWeldGun;
		MoveL [[-398.53,986.99,7.96],[0.390518,0.0535228,-0.919039,-0.00018247],[1,-1,1,0],[9E+09,9E+09,9E+09,9E+09,9E+09,9E+09]], vmax, z5, tWeldGun;
		ArcLStart [[-404.11,986.56,-9.77],[0.390535,0.0535541,-0.919029,-0.000151074],[1,-1,1,0],[9E+09,9E+09,9E+09,9E+09,9E+09,9E+09]], v20, seam13, weld13\Weave:=weave1, fine, tWeldGun;
		ArcL [[-404.10,964.74,-9.51],[0.390566,0.0535448,-0.919017,-0.000185269],[1,-1,1,0],[9E+09,9E+09,9E+09,9E+09,9E+09,9E+09]], v5, seam13, weld13\Weave:=weave1, z10, tWeldGun;
		ArcLEnd [[-428.88,950.30,-8.06],[0.237036,-0.623338,-0.70044,-0.254259],[1,-1,2,0],[9E+09,9E+09,9E+09,9E+09,9E+09,9E+09]], v5, seam13, weld13\Weave:=weave1, fine, tWeldGun;
		MoveL [[-432.86,900.19,113.28],[0.289357,-0.647919,-0.645007,-0.283619],[1,-1,2,0],[9E+09,9E+09,9E+09,9E+09,9E+09,9E+09]], vmax, z5, tWeldGun;
		MoveJ [[276.57,1109.67,795.31],[0.28935,-0.647904,-0.645024,-0.283623],[0,0,1,0],[9E+09,9E+09,9E+09,9E+09,9E+09,9E+09]], vmax, z5, tWeldGun;
	ENDPROC

PROC RunWeld(num i)

    MoveJ wp300{i}.trans, vmax, z50, tWeldGun;
    MoveJ wp300{i}.approach, vmax, z10, tWeldGun;
    MoveL wp300{i}.start, v50, z5, tWeldGun;
    ArcLStart wp300{i}.start, v5, wp300{i}.seamiii, wp300{i}.weldiii\Weave:=weave1, fine, tWeldGun;
    ArcLEnd   wp300{i}.end,   v5, wp300{i}.seamiii, wp300{i}.weldiii\Weave:=weave1, fine, tWeldGun;
    MoveL wp300{i}.exitt, v50, z5, tWeldGun;
ENDPROC


ENDMODULE
